PROGRAM PRG_Planning
VAR
    stMotionStage : ST_MotionStage;
    fbMotionAxisStageStepper : FB_MotionAXisStageStepper(
        MotionStage := stMotionStage
    );
END_VAR


fbMotionAxisStageStepper();

END_PROGRAM

(* stored: Version 1.1.0.1
   POU PRG_Planning: Id {f731b889-5613-47ef-a427-f056f64e7c91}, SpecialFunc None *)
